TYPE ST_LogLevelHeaders :
STRUCT
	Error	: STRING := '<Error> ';
	Warning	: STRING := '<Warning> ';
	Info	: STRING := '<Info> ';
END_STRUCT
END_TYPE

(* stored: Version 1.1.0.1, ProductVersion 3.1.4024.14
   DUT ST_LogLevelHeaders: Id {f8a141c0-97a4-0344-3fb2-17e7c83e461f} *)
